# EPICS substitutions: db/Beckhoff_5XXX/ecmcEL5131_DC.substitutions
file "ecmcEL5131-chX.template"
{
    pattern {CH_ID}
            {01   }

}

# timestamp
file "ecmc_timestamp_64-chX.template"{
  pattern {CH_ID, KEY,      suffix,        sourceName          }
          {"",    "Enc01",  "-Time",       "timestamp01"       }
          {"",    "Enc01",  "-TimeIdx",    "timestampIndex01"  }
          {"",    "Enc01",  "-TimeLtch01", "timestampLatch01"  }
          {"",    "Enc01",  "-TimeLtch02", "timestampLatch02"  }
}
